// Mitsubishi GX Works2 project: BookEX6_9 Limit   PLC: Q13UDV

// global labels: Global
VAR_GLOBAL
  bVar0 AT M5000 : BOOL;
  abArray0 AT M5010 : ARRAY [0..49] OF BOOL;
  sStr0 AT D5000 : STRING[199];
  sStr1 AT D5100 : STRING[199];
  sStr2 AT D5200 : STRING[199];
  sStr3 AT D5300 : STRING[199];
  sStr4 AT D5400 : STRING[199];
  sStr5 AT D5500 : STRING[199];
  sStr6 AT D5600 : STRING[199];
  sStr7 AT D5700 : STRING[199];
  sStr8 AT D5800 : STRING[199];
  sStr9 AT D5900 : STRING[199];
  iVar0 AT D4500 : INT;
  iVar1 AT D4501 : INT;
  iVar2 AT D4502 : INT;
  iVar3 AT D4503 : INT;
  iVar4 AT D4504 : INT;
  iVar5 AT D4505 : INT;
  iVar6 AT D4506 : INT;
  iVar7 AT D4507 : INT;
  iVar8 AT D4508 : INT;
  iVar9 AT D4509 : INT;
  dVar0 AT D4510 : DINT;
  dVar1 AT D4512 : DINT;
  dVar2 AT D4514 : DINT;
  dVar3 AT D4516 : DINT;
  dVar4 AT D4518 : DINT;
  dVar5 AT D4520 : DINT;
  dVar6 AT D4522 : DINT;
  dVar7 AT D4524 : DINT;
  dVar8 AT D4526 : DINT;
  dVar9 AT D4528 : DINT;
  wVar0 AT D4530 : WORD;
  wVar1 AT D4531 : WORD;
  wVar2 AT D4532 : WORD;
  wVar3 AT D4533 : WORD;
  wVar4 AT D4534 : WORD;
  wVar5 AT D4535 : WORD;
  wVar6 AT D4536 : WORD;
  wVar7 AT D4537 : WORD;
  wVar8 AT D4538 : WORD;
  wVar9 AT D4539 : WORD;
  dwVar0 AT D4540 : DWORD;
  dwVar1 AT D4542 : DWORD;
  dwVar2 AT D4544 : DWORD;
  dwVar3 AT D4546 : DWORD;
  dwVar4 AT D4548 : DWORD;
  dwVar5 AT D4550 : DWORD;
  dwVar6 AT D4552 : DWORD;
  dwVar7 AT D4554 : DWORD;
  dwVar8 AT D4556 : DWORD;
  dwVar9 AT D4558 : DWORD;
  fsVar0 AT D4560 : REAL;
  fsVar1 AT D4562 : REAL;
  fsVar2 AT D4564 : REAL;
  fsVar3 AT D4566 : REAL;
  fsVar4 AT D4568 : REAL;
  fsVar5 AT D4570 : REAL;
  fsVar6 AT D4572 : REAL;
  fsVar7 AT D4574 : REAL;
  fsVar8 AT D4576 : REAL;
  fsVar9 AT D4578 : REAL;
  fdVar0 AT D4580 : LREAL;
  tTime0 AT D4620 : TIME;
  tTime1 AT D4622 : TIME;
  tTime2 AT D4624 : TIME;
  tTime3 AT D4626 : TIME;
  tTime4 AT D4628 : TIME;
  tTime5 AT D4630 : TIME;
  tTime6 AT D4632 : TIME;
  tTime7 AT D4634 : TIME;
  tTime8 AT D4636 : TIME;
  tTime9 AT D4638 : TIME;
  tTime10 AT D4640 : TIME;
  bVar1 AT M5001 : BOOL;
  bVar2 AT M5002 : BOOL;
  bVar3 AT M5003 : BOOL;
  bVar4 AT M5004 : BOOL;
  bVar5 AT M5005 : BOOL;
  bVar6 AT M5006 : BOOL;
  bVar7 AT M5007 : BOOL;
  bVar8 AT M5008 : BOOL;
  bVar9 AT M5009 : BOOL;
  abArray1 AT M5060 : ARRAY [0..49] OF BOOL;
  abArray2 AT M5110 : ARRAY [0..49] OF BOOL;
  abArray3 AT M5160 : ARRAY [0..49] OF BOOL;
  abArray4 AT M5210 : ARRAY [0..49] OF BOOL;
  abArray5 AT M5260 : ARRAY [0..49] OF BOOL;
  abArray6 AT M5310 : ARRAY [0..49] OF BOOL;
  abArray7 AT M5360 : ARRAY [0..49] OF BOOL;
  abArray8 AT M5410 : ARRAY [0..49] OF BOOL;
  abArray9 AT M5460 : ARRAY [0..49] OF BOOL;
  fdVar1 AT D4584 : LREAL;
  fdVar2 AT D4588 : LREAL;
  fdVar3 AT D4592 : LREAL;
  fdVar4 AT D4596 : LREAL;
  fdVar5 AT D4600 : LREAL;
  fdVar6 AT D4604 : LREAL;
  fdVar7 AT D4608 : LREAL;
  fdVar8 AT D4612 : LREAL;
  fdVar9 AT D4616 : LREAL;
END_VAR
// user libraries (not included): HMI

FUNCTION INV_REAL
VAR_INPUT
  fs_V : REAL;
END_VAR
;
IF fs_V <> 0.0 THEN 
	INV_REAL := 1.0 / fs_V; 
END_IF;
END_FUNCTION

FUNCTION MID_REAL
VAR_INPUT
  fs_IN1 : REAL;
  fs_IN2 : REAL;
  fs_IN3 : REAL;
END_VAR
VAR
  fsD1 : REAL;
  fsD2 : REAL;
  fsD3 : REAL;
  fsTmp : REAL;
END_VAR
;
fsD1 := fs_IN1;
fsD2 := fs_IN2;
fsD3 := fs_IN3;
IF fsD1 > fsD2 THEN 
	fsTmp := fsD1; 
	fsD1 := fsD2; 
	fsD2 := fsTmp; 
END_IF;
IF fsD2 > fsD3 THEN 
	fsD2 := fsD3; 
END_IF;
MID_REAL := SEL(fsD1 > fsD2, fsD2, fsD1);
END_FUNCTION

FUNCTION MUX_REAL2
VAR_INPUT
  fs_IN0 : REAL;
  fs_IN1 : REAL;
  b_S : BOOL;
END_VAR
;
MUX_REAL2 := SEL(b_S, fs_IN0, fs_IN1);
END_FUNCTION

FUNCTION MUX_REAL4
VAR_INPUT
  fs_IN0 : REAL;
  fs_IN1 : REAL;
  b_S0 : BOOL;
  b_S1 : BOOL;
  fs_IN2 : REAL;
  fs_IN3 : REAL;
END_VAR
;
IF b_S1 THEN
	MUX_REAL4 := SEL(b_S0, fs_IN2, fs_IN3);
ELSE
	MUX_REAL4 := SEL(b_S0, fs_IN0, fs_IN1);
END_IF;
END_FUNCTION

FUNCTION SIGN_REAL
VAR_INPUT
  fs_V : REAL;
END_VAR
;
IF fs_V > 0.0 THEN
	SIGN_REAL := 1;
ELSIF fs_V < 0.0 THEN
	SIGN_REAL := -1;
ELSE
	SIGN_REAL := 0;
END_IF;
END_FUNCTION

PROGRAM ExLIMITATION
VAR
  Var_D0 : WORD;
  Var_D1 : INT;
END_VAR
(* structured ladder/FBD written out as ST: instructions are called as NAME(EN, inputs, outputs); _pN, _eN, _tN stand for wires *)
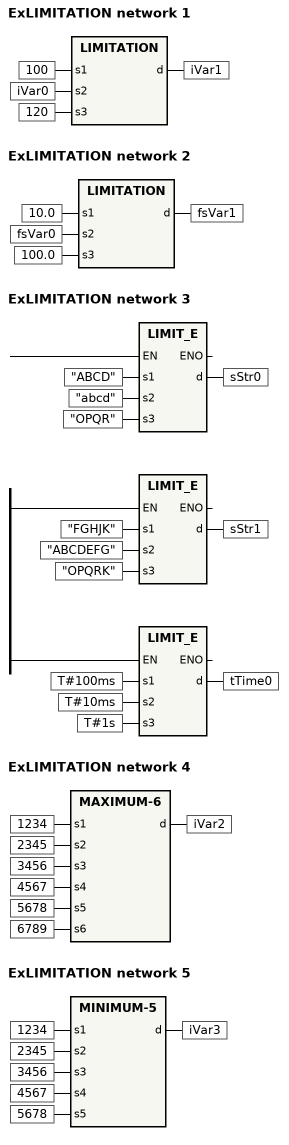
(* network 1 *)
iVar1 := LIMITATION(100, iVar0, 120);
(* network 2 *)
fsVar1 := LIMITATION(10.0, fsVar0, 100.0);
(* network 3 *)
LIMIT_E(TRUE, "ABCD", "abcd", "OPQR", sStr0);
LIMIT_E(TRUE, "FGHJK", "ABCDEFG", "OPQRK", sStr1);
LIMIT_E(TRUE, T#100ms, T#10ms, T#1s, tTime0);
(* network 4 *)
iVar2 := MAXIMUM(1234, 2345, 3456, 4567, 5678, 6789);
(* network 5 *)
iVar3 := MINIMUM(1234, 2345, 3456, 4567, 5678);
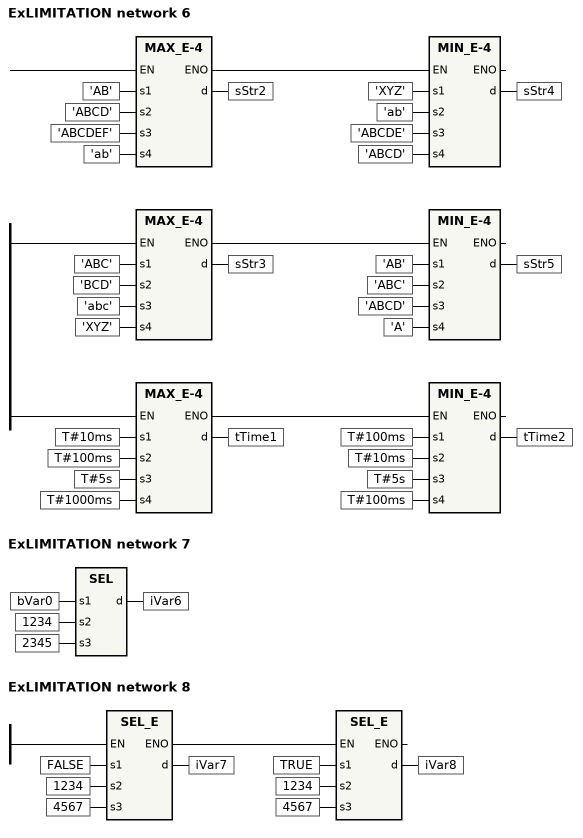
(* network 6 *)
_e1 := MAX_E(TRUE, 'AB', 'ABCD', 'ABCDEF', 'ab', sStr2);
MIN_E(_e1, 'XYZ', 'ab', 'ABCDE', 'ABCD', sStr4);
_e2 := MAX_E(TRUE, 'ABC', 'BCD', 'abc', 'XYZ', sStr3);
MIN_E(_e2, 'AB', 'ABC', 'ABCD', 'A', sStr5);
_e3 := MAX_E(TRUE, T#10ms, T#100ms, T#5s, T#1000ms, tTime1);
MIN_E(_e3, T#100ms, T#10ms, T#5s, T#100ms, tTime2);
(* network 7 *)
iVar6 := SEL(bVar0, 1234, 2345);
(* network 8 *)
_e1 := SEL_E(TRUE, FALSE, 1234, 4567, iVar7);
SEL_E(_e1, TRUE, 1234, 4567, iVar8);
END_PROGRAM

PROGRAM ExMID
(* structured ladder/FBD written out as ST: instructions are called as NAME(EN, inputs, outputs); _pN, _eN, _tN stand for wires *)
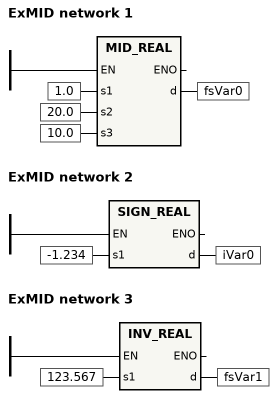
(* network 1 *)
MID_REAL(TRUE, 1.0, 20.0, 10.0, fsVar0);
(* network 2 *)
SIGN_REAL(TRUE, -1.234, iVar0);
(* network 3 *)
INV_REAL(TRUE, 123.567, fsVar1);
END_PROGRAM

PROGRAM ExMUX_REAL
(* structured ladder/FBD written out as ST: instructions are called as NAME(EN, inputs, outputs); _pN, _eN, _tN stand for wires *)
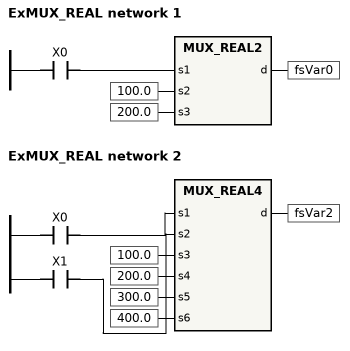
(* network 1 *)
fsVar0 := MUX_REAL2(X0, 100.0, 200.0);
(* network 2 *)
fsVar2 := MUX_REAL4(X0, X1, 100.0, 200.0, 300.0, 400.0);
END_PROGRAM

PROGRAM ExMUX
VAR
  bAutoMode : BOOL;
  bManMode : BOOL;
  tDelayTime : TIME;
END_VAR
(* structured ladder/FBD written out as ST: instructions are called as NAME(EN, inputs, outputs); _pN, _eN, _tN stand for wires *)
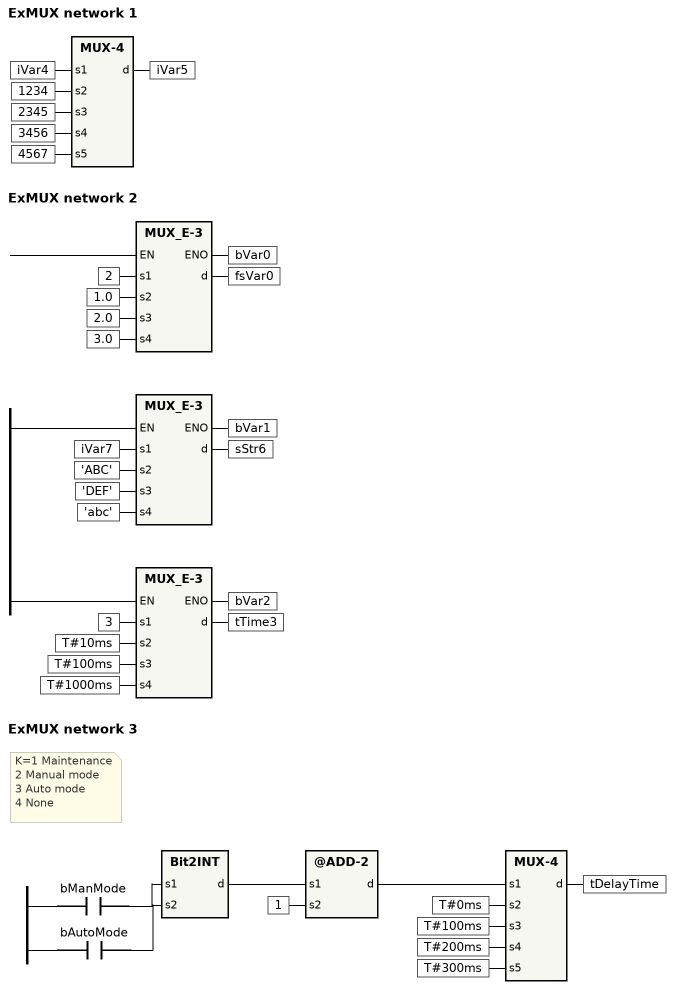
(* network 1 *)
iVar5 := MUX(iVar4, 1234, 2345, 3456, 4567);
(* network 2 *)
_e1 := MUX_E(TRUE, 2, 1.0, 2.0, 3.0, fsVar0);
bVar0 := _e1;
_e2 := MUX_E(TRUE, iVar7, 'ABC', 'DEF', 'abc', sStr6);
bVar1 := _e2;
_e3 := MUX_E(TRUE, 3, T#10ms, T#100ms, T#1000ms, tTime3);
bVar2 := _e3;
(* network 3 *)
(* K=1 Maintenance /      2 Manual mode /      3 Auto mode /      4 None *)
tDelayTime := MUX(@ADD-2(Bit2INT(bManMode, bAutoMode), 1), T#0ms, T#100ms, T#200ms, T#300ms);
END_PROGRAM

FUNCTION Bit2INT
VAR_INPUT
  Bit0 : BOOL;
  Bit1 : BOOL;
END_VAR
;
Bit2INT := BOOL_TO_INT(Bit0) * 1 + BOOL_TO_INT(Bit1) * 2;
END_FUNCTION

PROGRAM ExLimit_ST
VAR
  bCalcOK : BOOL;
  bEnable : BOOL;
  HmiSpd : INT;
  MotorSpd : INT;
  bCalcError : BOOL;
END_VAR
;

(* LIMITATION_E 함수 호출 및 입력변수 *)
bCalcOK := LIMIT_E(TRUE, 100, HmiSpd, 3000, MotorSpd);

(* ENO  활용한 에러 진단 인터록 추가 *)
IF bEnable AND NOT bCalcOK THEN 
	bCalcError := TRUE; 	(* 명령 에러 시 알람 발생 *)
ELSE 
	bCalcError := FALSE; 
END_IF;
END_PROGRAM

PROGRAM ExMin_Max
VAR
  Min_Max_1 : Min_Max;
END_VAR
(* structured ladder/FBD written out as ST: instructions are called as NAME(EN, inputs, outputs); _pN, _eN, _tN stand for wires *)
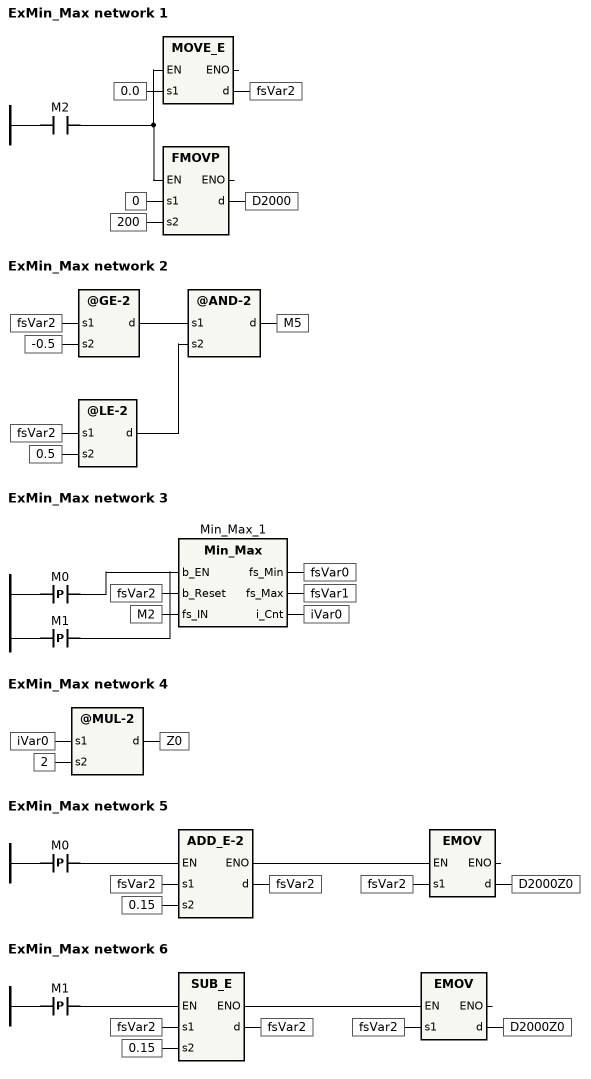
(* network 1 *)
MOVE_E(M2, 0.0, fsVar2);
FMOVP(M2, 0, 200, D2000);
(* network 2 *)
M5 := @AND-2(@GE-2(fsVar2, -0.5), @LE-2(fsVar2, 0.5));
(* network 3 *)
Min_Max_1(b_EN := LDP(TRUE, M0) OR LDP(TRUE, M1), b_Reset := fsVar2, fs_IN := M2, fs_Min => fsVar0, fs_Max => fsVar1, i_Cnt => iVar0);
(* network 4 *)
Z0 := @MUL-2(iVar0, 2);
(* network 5 *)
_e1 := ADD_E(LDP(TRUE, M0), fsVar2, 0.15, fsVar2);
EMOV(_e1, fsVar2, D2000Z0);
(* network 6 *)
_e1 := SUB_E(LDP(TRUE, M1), fsVar2, 0.15, fsVar2);
EMOV(_e1, fsVar2, D2000Z0);
END_PROGRAM

FUNCTION_BLOCK Min_Max
VAR_INPUT
  b_EN : BOOL;
  b_Reset : BOOL;
END_VAR
VAR_OUTPUT
  fs_Min : REAL;
  fs_Max : REAL;
  i_Cnt : INT;
END_VAR
VAR_INPUT
  fs_IN : REAL;
END_VAR
;
IF b_Reset THEN
	fs_Min := fs_IN;
	fs_Max := fs_IN;
	i_Cnt := 0;
ELSIF b_EN THEN
	i_Cnt := i_Cnt+1;
	IF fs_IN < fs_Min THEN fs_Min := fs_IN;  
	ELSIF fs_IN > fs_Max THEN fs_Max := fs_IN;  
	END_IF;
END_IF;
END_FUNCTION_BLOCK
